	                #CambioReqVel := "Motore".M[#K_MotoreInt].Dati.VeloRichPerc <> "Motore".M[#K_MotoreInt].In.CmdVelocitaRich;
	                IF #CambioReqVel THEN
	                    "Motore".M[#K_MotoreInt].Dati.VeloRichPerc := "Motore".M[#K_MotoreInt].In.CmdVelocitaRich;
	                END_IF;
	(* Controllo Cambio Accelerazione richiesta *)
	                #CambioReqAcc := "Motore".M[#K_MotoreInt].Dati.AccRichPerc <> "Motore".M[#K_MotoreInt].In.Acc;
	                IF #CambioReqAcc THEN
	                    "Motore".M[#K_MotoreInt].Dati.AccRichPerc := "Motore".M[#K_MotoreInt].In.Acc;
	                END_IF;
	(* Controllo Cambio Decelerazione richiesta *)
	                #CambioReqDec := "Motore".M[#K_MotoreInt].Dati.DecRichPerc <> "Motore".M[#K_MotoreInt].In.Dec;
	                IF #CambioReqDec THEN
	                    "Motore".M[#K_MotoreInt].Dati.DecRichPerc := "Motore".M[#K_MotoreInt].In.Dec;
	                END_IF;
	            END_REGION
	            REGION Direzione Movimento Richiesta
	                IF "Motore".M[#K_MotoreInt].In.CmdPosRich AND "Motore".M[#K_MotoreInt].Out.Pronto AND #AbilDirPos THEN
	                    #ReqDirPos := TRUE;
	                    #ReqDirNeg := FALSE;
	                    #UnaDirezioneRichiesta := TRUE;
	                ELSIF "Motore".M[#K_MotoreInt].In.CmdNegRich AND "Motore".M[#K_MotoreInt].Out.Pronto AND #AbilDirNeg THEN
	                    #ReqDirPos := FALSE;
	                    #ReqDirNeg := TRUE;
	                    #UnaDirezioneRichiesta := TRUE;
	                ELSE
	                    #ReqDirPos := FALSE;
	                    #ReqDirNeg := FALSE;
	                    #UnaDirezioneRichiesta := FALSE;
	                END_IF;
	            END_REGION
	        END_IF;
	    END_REGION ;
	    REGION Parameter profile
	        REGION VelocitÃ  Minima
	            IF NOT "Motore".M[#K_MotoreInt].Dati.ActVelPos AND NOT "Motore".M[#K_MotoreInt].Dati.ActVelNeg AND #ReqDirNeg OR "Motore".M[#K_MotoreInt].Dati.ActVelNeg THEN
	                #SpazioFrenoDir := "Motore".M[#K_MotoreInt].Prm.SpazioArrestoNeg;
	                #VeloFrenoDir := "Motore".M[#K_MotoreInt].Prm.VelSgancioFrenoNeg;
	            ELSE
	                #SpazioFrenoDir := "Motore".M[#K_MotoreInt].Prm.SpazioArrestoPos;
	                #VeloFrenoDir := "Motore".M[#K_MotoreInt].Prm.VelSgancioFrenoPos;
	            END_IF;
	        END_REGION
	        REGION Controllo VelocitÃ
	(* Controllo che la velocitÃ  sia all'interno del limite Sgancio Freno < VeloRich < VeloMax *)
	            "Motore".M[#K_MotoreInt].Allarmi.TrgVelMinFreno := false;
	            "Motore".M[#K_MotoreInt].Allarmi.TrgVelMaxMax := false;
	            "Motore".M[#K_MotoreInt].Allarmi.TrgVelCamMinFreno := false;
	            "Motore".M[#K_MotoreInt].Allarmi.TrgVelCamMaxMax := false;
	            IF #UnaDirezioneRichiesta THEN
	                IF "Motore".M[#K_MotoreInt].Dati.VeloRichPerc < #VeloFrenoDir THEN
	                    "Motore".M[#K_MotoreInt].Allarmi.TrgVelMinFreno := true;
	                    "Motore".M[#K_MotoreInt].Allarmi.Parametri := TRUE;
	                    "Motore".M[#K_MotoreInt].Dati.VeloRichPerc := #VeloFrenoDir;
	                END_IF;
	                IF "Motore".M[#K_MotoreInt].Dati.VeloRichPerc > "Motore".M[#K_MotoreInt].Prm.C.VelMax THEN
	                    "Motore".M[#K_MotoreInt].Allarmi.TrgVelMaxMax := true;
	                    "Motore".M[#K_MotoreInt].Allarmi.Parametri := TRUE;
	                    "Motore".M[#K_MotoreInt].Dati.VeloRichPerc := "Motore".M[#K_MotoreInt].Prm.C.VelMax;
	                END_IF;
	                (* Controllo che la velocitÃ  di cambio VelocitÃ  sia all'interno del limite Sgancio Freno < VeloRich < VeloMax *)
	                IF "Motore".M[#K_MotoreInt].In.CambioVelDaPunto THEN
	                    "Motore".M[#K_MotoreInt].Dati.VeloDopoCambioRich := "Motore".M[#K_MotoreInt].In.VelCambioVel;
	                    IF "Motore".M[#K_MotoreInt].Dati.VeloDopoCambioRich < #VeloFrenoDir THEN
	                        "Motore".M[#K_MotoreInt].Allarmi.TrgVelCamMinFreno := true;
	                        "Motore".M[#K_MotoreInt].Allarmi.Parametri := TRUE;
	                        "Motore".M[#K_MotoreInt].Dati.VeloDopoCambioRich := #VeloFrenoDir;
	                    END_IF;
	                    IF "Motore".M[#K_MotoreInt].Dati.VeloDopoCambioRich > "Motore".M[#K_MotoreInt].Prm.C.VelMax THEN
	                        "Motore".M[#K_MotoreInt].Allarmi.TrgVelCamMaxMax := true;
	                        "Motore".M[#K_MotoreInt].Allarmi.Parametri := TRUE;
	                        "Motore".M[#K_MotoreInt].Dati.VeloDopoCambioRich := "Motore".M[#K_MotoreInt].Prm.C.VelMax;
	                    END_IF;
	                END_IF;
	            END_IF;
	        END_REGION
	        REGION Controllo Decelerazione di emergenza
	            IF "Motore".M[#K_MotoreInt].Dati.Memo_Req_Dec_Emergenza <> "Motore".M[#K_MotoreInt].Prm.DecEmergenza THEN
	                "Motore".M[#K_MotoreInt].Allarmi.DecEmergenzaRichZero := "Motore".M[#K_MotoreInt].Prm.DecEmergenza < 100;
	                IF "Motore".M[#K_MotoreInt].Allarmi.DecEmergenzaRichZero THEN
	                    "Motore".M[#K_MotoreInt].Dati.Memo_Req_Dec_Emergenza := 100;
	                    "Motore".M[#K_MotoreInt].Allarmi.Parametri := TRUE;
	                    #CambioReqAcc := true;
	                    #CambioReqDec := true;
	                ELSE
	                    "Motore".M[#K_MotoreInt].Dati.Memo_Req_Dec_Emergenza := "Motore".M[#K_MotoreInt].Prm.DecEmergenza;
	                END_IF;
	            END_IF;
	        END_REGION
	        REGION Controllo Decelerazione
	            IF #CambioReqDec THEN
	                "Motore".M[#K_MotoreInt].Allarmi.DecRichZero := "Motore".M[#K_MotoreInt].Dati.DecRichPerc < 100;
	                IF "Motore".M[#K_MotoreInt].Allarmi.DecRichZero THEN
	                    "Motore".M[#K_MotoreInt].Dati.DecRichPerc := 100;
	                    "Motore".M[#K_MotoreInt].Allarmi.Parametri := TRUE;
	                END_IF;
	                "Motore".M[#K_MotoreInt].Allarmi.DecRichMaxMaxDec := "Motore".M[#K_MotoreInt].Dati.DecRichPerc > "Motore".M[#K_MotoreInt].Dati.Memo_Req_Dec_Emergenza;
	                IF "Motore".M[#K_MotoreInt].Allarmi.DecRichMaxMaxDec THEN
	                    "Motore".M[#K_MotoreInt].Dati.DecRichPerc := "Motore".M[#K_MotoreInt].Dati.Memo_Req_Dec_Emergenza;
	                    "Motore".M[#K_MotoreInt].Allarmi.Parametri := TRUE;
	                END_IF;
	            END_IF;
	        END_REGION
	        REGION Controllo Decelerazione Finale
	            "Motore".M[#K_MotoreInt].Allarmi.DecFinaleRichZero := "Motore".M[#K_MotoreInt].Prm.DecFinale < 100;
	            IF "Motore".M[#K_MotoreInt].Allarmi.DecFinaleRichZero THEN
	                "Motore".M[#K_MotoreInt].Prm.DecFinale := 100;
	                "Motore".M[#K_MotoreInt].Allarmi.Parametri := TRUE;
	            END_IF;
	            "Motore".M[#K_MotoreInt].Allarmi.DecFinaleRichMaxMaxDec := "Motore".M[#K_MotoreInt].Prm.DecFinale > "Motore".M[#K_MotoreInt].Dati.Memo_Req_Dec_Emergenza;
	            IF "Motore".M[#K_MotoreInt].Allarmi.DecFinaleRichMaxMaxDec THEN
	                "Motore".M[#K_MotoreInt].Prm.DecFinale := "Motore".M[#K_MotoreInt].Dati.Memo_Req_Dec_Emergenza;
	                "Motore".M[#K_MotoreInt].Allarmi.Parametri := TRUE;
	            END_IF;
	            IF "Motore".M[#K_MotoreInt].Prm.DecFinale <> "Motore".M[#K_MotoreInt].Dati.DecReqFinaleInLavo THEN
	                IF NOT "Motore".M[#K_MotoreInt].Out.InMarcia OR "Motore".M[#K_MotoreInt].Prm.DecFinale > "Motore".M[#K_MotoreInt].Dati.DecReqFinaleInLavo THEN
	                    "Motore".M[#K_MotoreInt].Dati.DecReqFinaleInLavo := "Motore".M[#K_MotoreInt].Prm.DecFinale;
	                END_IF;
	            END_IF;
	        END_REGION
	        REGION Controllo Accelerazione
	            IF #CambioReqAcc THEN
	                "Motore".M[#K_MotoreInt].Allarmi.AccRichZero := "Motore".M[#K_MotoreInt].Dati.AccRichPerc < 100;
	                IF "Motore".M[#K_MotoreInt].Allarmi.AccRichZero THEN
	                    "Motore".M[#K_MotoreInt].Dati.AccRichPerc := 100;
	                    "Motore".M[#K_MotoreInt].Allarmi.Parametri := TRUE;
	                END_IF;
	                "Motore".M[#K_MotoreInt].Allarmi.AccRichMaxMaxDec := "Motore".M[#K_MotoreInt].Dati.AccRichPerc > "Motore".M[#K_MotoreInt].Dati.Memo_Req_Dec_Emergenza;
	                IF "Motore".M[#K_MotoreInt].Allarmi.AccRichMaxMaxDec THEN
	                    "Motore".M[#K_MotoreInt].Dati.AccRichPerc := "Motore".M[#K_MotoreInt].Dati.Memo_Req_Dec_Emergenza;
	                    "Motore".M[#K_MotoreInt].Allarmi.Parametri := TRUE;
	                END_IF;
	            END_IF;
	        END_REGION
	        REGION Assegnazione decelerazione
	            IF "Motore".M[#K_MotoreInt].Dati.DecRichPerc <> "Motore".M[#K_MotoreInt].Dati.DecReqInLavo THEN
	                IF NOT "Motore".M[#K_MotoreInt].Out.InMarcia OR "Motore".M[#K_MotoreInt].Dati.DecRichPerc > "Motore".M[#K_MotoreInt].Dati.DecReqInLavo OR "Motore".M[#K_MotoreInt].Out.VelAss < #VeloBassaConv THEN
	                    "Motore".M[#K_MotoreInt].Dati.DecReqInLavo := "Motore".M[#K_MotoreInt].Dati.DecRichPerc;
	                END_IF;
	            END_IF;
	        END_REGION
	        REGION Assegnazione decelerazione D'emergenza
	            IF "Motore".M[#K_MotoreInt].Dati.Memo_Req_Dec_Emergenza <> "Motore".M[#K_MotoreInt].Dati.DecReqEmergInLavo THEN
	                IF NOT "Motore".M[#K_MotoreInt].Out.InMarcia OR "Motore".M[#K_MotoreInt].Dati.Memo_Req_Dec_Emergenza > "Motore".M[#K_MotoreInt].Dati.DecReqEmergInLavo THEN
	                    "Motore".M[#K_MotoreInt].Dati.DecReqEmergInLavo := "Motore".M[#K_MotoreInt].Dati.Memo_Req_Dec_Emergenza;
	                END_IF;
	            END_IF;
	        END_REGION
	        REGION Calcolo Lo Spazio Di Arresto
	            #ReqDecBassa := FALSE;
	            #ReqDecStop := FALSE;
	            #BloccaAcc := FALSE;
	            IF "Motore".M[#K_MotoreInt].Out.InMarcia THEN
	                IF "Motore".M[#K_MotoreInt].Out.VelAss > #VeloBassaConv THEN
	                    #SpazioStop_01 := (SQR(IN := "Motore".M[#K_MotoreInt].Out.VelAss) - SQR(IN := #VeloBassaConv)) / DINT_TO_REAL("Motore".M[#K_MotoreInt].Dati.DecReqInLavo) / 2.0;
	                    #SpazioStop_02 := DINT_TO_REAL(IN := "Motore".M[#K_MotoreInt].Prm.TBassaVel) * #VeloBassaConv / 1000.0;
	                    #SpazioStop_03 := (SQR(IN := #VeloBassaConv) - SQR(IN := DINT_TO_REAL(#VeloFrenoDir))) / DINT_TO_REAL("Motore".M[#K_MotoreInt].Dati.DecReqFinaleInLavo) / 2.0;
	                ELSE
	                    #SpazioStop_01 := 0.0;
	                    #SpazioStop_02 := 0.0;
	                    #SpazioStop_03 := (SQR(IN := "Motore".M[#K_MotoreInt].Out.VelAss) - SQR(IN := DINT_TO_REAL(#VeloFrenoDir))) / DINT_TO_REAL("Motore".M[#K_MotoreInt].Dati.DecReqFinaleInLavo) / 2.0;
	                    ;
	                END_IF;
	                #SpazioStop_04 := INT_TO_REAL("Motore".M[#K_MotoreInt].Prm.TReazioneSistema) * ("Motore".M[#K_MotoreInt].Out.VelAss - DINT_TO_REAL(#VeloFrenoDir)) / 1000.0;
	                #SpazioStop := TRUNC(IN := #SpazioStop_03 + #SpazioStop_04) + #SpazioFrenoDir;
	                #SpazioBassa := TRUNC(IN := #SpazioStop_01 + #SpazioStop_02) + #SpazioStop;
	                IF #FunzPositioning THEN
	                    #BloccaAcc := TRUNC(("Motore".M[#K_MotoreInt].Out.VelAss * INT_TO_REAL("Motore".M[#K_MotoreInt].Prm.TMinVCost) / 1000.0)) + #SpazioStop > #DistTRG_ASS;
	                    #ReqDecBassa := #DistTRG_ASS < #SpazioBassa;
	                    #ReqDecStop := #DistTRG_ASS < #SpazioStop;
	                END_IF;
	            ELSE
	                #SpazioBassa := #SpazioStop := #SpazioFrenoDir;
	            END_IF;
	        END_REGION
	        REGION Calcolo lo spazio passaggio seconda Vel.
	            IF #FunzPositioning AND "Motore".M[#K_MotoreInt].In.CambioVelDaPunto AND NOT "Motore".M[#K_MotoreInt].Dati.MotoreFermo THEN
	                // Lo spazio di cambio velocitÃ  Ã¨ dato dalla somma dei seguenti fattori:

	                // 1) Spazio necessario al cambio velocitÃ  dell'asse calcolando una rampa trapezoidale.
	                // 2) Simulazione dello spazio percorso dall'asse durante la reazione del segnale analogico.

	                // Condizione 01 -Trapezio passaggio dalla velocitÃ  di lavoro alla velocitÃ  bassa
	                #SpazioCambioVel_01 := ("Motore".M[#K_MotoreInt].Out.VelAss ** 2 - DINT_TO_REAL("Motore".M[#K_MotoreInt].Dati.VeloDopoCambioRich) ** 2) / DINT_TO_REAL("Motore".M[#K_MotoreInt].Dati.DecReqInLavo) / 2.0;
	                #SpazioCambioVel_02 := INT_TO_REAL("Motore".M[#K_MotoreInt].Prm.TReazioneSistema) * "Motore".M[#K_MotoreInt].Out.VelAss / 1000.0;
	                #SpazioCambioVel := TRUNC(#SpazioCambioVel_01 + #SpazioCambioVel_02);
	                // Continua solo se cambio velocitÃ  Ã¨ attivo
	                // Calcolo la distanza dal cambio velocitÃ
	                IF NOT "Motore".M[#K_MotoreInt].In.PosRelativo THEN
	                    IF "Motore".M[#K_MotoreInt].Prm.Mech.EndLess THEN
	                        WHILE "Motore".M[#K_MotoreInt].In.PosCambioVel > "Motore".M[#K_MotoreInt].Prm.Enc.ModuloPosEnc DO
	                            "Motore".M[#K_MotoreInt].In.PosCambioVel -= #RicircoloTotale;
	                        END_WHILE;
	                        WHILE "Motore".M[#K_MotoreInt].In.PosCambioVel < "Motore".M[#K_MotoreInt].Prm.Enc.ModuloNegEnc DO
	                            "Motore".M[#K_MotoreInt].In.PosCambioVel += #RicircoloTotale;
	                        END_WHILE;
	                    END_IF;
	                    IF "Motore".M[#K_MotoreInt].Dati.ActVelPos THEN
	                        #DistCambioVel := "Motore".M[#K_MotoreInt].Out.ActPos + #SpazioCambioVel - "Motore".M[#K_MotoreInt].In.PosCambioVel;
	                    ELSE
	                        #DistCambioVel := "Motore".M[#K_MotoreInt].Out.ActPos - #SpazioCambioVel - "Motore".M[#K_MotoreInt].In.PosCambioVel;
	                    END_IF;
	                    IF "Motore".M[#K_MotoreInt].Prm.Mech.EndLess THEN
	                        IF #DistCambioVel > #MezzoRicircoloTotale THEN
	                            #DistCambioVel -= #RicircoloTotale;
	                        END_IF;
	                        IF #DistCambioVel < - #MezzoRicircoloTotale THEN
	                            #DistCambioVel += #RicircoloTotale;
	                        END_IF;
	                    END_IF;
	                    #ReqCambioVel := #DistCambioVel >= 0 AND "Motore".M[#K_MotoreInt].Dati.ActVelPos OR #DistCambioVel < 0 AND "Motore".M[#K_MotoreInt].Dati.ActVelNeg;
	                ELSE
	                    #ReqCambioVel := "Motore".M[#K_MotoreInt].Dati.MovRelRichiesto - #DistTRG_ASS + #SpazioCambioVel > "Motore".M[#K_MotoreInt].In.PosCambioVel;
	                END_IF;
	            ELSE
	                #ReqCambioVel := FALSE;
	                #SpazioCambioVel := 0;
	            END_IF;

	        END_REGION
	        REGION Pos.Motore + Spazio Arresto
	            IF "Motore".M[#K_MotoreInt].Out.InMarcia THEN
	                "Motore".M[#K_MotoreInt].Out.SpazioStop := #SpazioBassa;
	                IF "Motore".M[#K_MotoreInt].Dati.ActVelPos THEN
	                    "Motore".M[#K_MotoreInt].Out.ActPosPiuStop := "Motore".M[#K_MotoreInt].Out.ActPos + #SpazioBassa;
	                ELSE
	                    "Motore".M[#K_MotoreInt].Out.ActPosPiuStop := "Motore".M[#K_MotoreInt].Out.ActPos - #SpazioBassa;
	                END_IF;
	                IF "Motore".M[#K_MotoreInt].Prm.Mech.EndLess THEN
	                    IF "Motore".M[#K_MotoreInt].Out.ActPosPiuStop < "Motore".M[#K_MotoreInt].Prm.Enc.ModuloNegEnc THEN
	                        "Motore".M[#K_MotoreInt].Out.ActPosPiuStop += #RicircoloTotale;
	                    END_IF;
	                    IF "Motore".M[#K_MotoreInt].Out.ActPosPiuStop > "Motore".M[#K_MotoreInt].Prm.Enc.ModuloPosEnc THEN
	                        "Motore".M[#K_MotoreInt].Out.ActPosPiuStop -= #RicircoloTotale;
	                    END_IF;
	                END_IF;
	            ELSE
	                "Motore".M[#K_MotoreInt].Out.ActPosPiuStop := "Motore".M[#K_MotoreInt].Out.ActPos;
	                "Motore".M[#K_MotoreInt].Out.SpazioStop := 0;
	            END_IF;
	        END_REGION
	    END_REGION ;
	    REGION Delay brake
	        REGION Ritrado Aggancio/Sgancio Freno
	            IF "Motore".M[#K_MotoreInt].Prm.FrenoPresente THEN
	                IF "Motore".M[#K_MotoreInt].Prm.FBKFrenoPresente THEN
	                    "Motore".M[#K_MotoreInt].Dati.StatoFreno := "Motore".M[#K_MotoreInt].In.FrenoSganciato;
	                ELSE
	                    "Motore".M[#K_MotoreInt].Dati.StatoFreno := "Motore".M[#K_MotoreInt].Out.CmdFreno;
	                END_IF;
	                IF "Motore".M[#K_MotoreInt].Dati.StatoFreno THEN
	                    "Motore".M[#K_MotoreInt].Dati.ContAggancioFreno := 0;
	                    "Motore".M[#K_MotoreInt].Dati.RitAggancioFreno := false;
	                    IF NOT "Motore".M[#K_MotoreInt].Out.RitSgancioFreno THEN
	                        "Motore".M[#K_MotoreInt].Out.RitSgancioFreno := "Motore".M[#K_MotoreInt].Dati.ContSgancioFreno >= "Motore".M[#K_MotoreInt].Prm.TSgancioFreno;
	                        "Motore".M[#K_MotoreInt].Dati.ContSgancioFreno += REAL_TO_INT("Zona".Comuni.TempoCicloCpu_r);
	                    END_IF;
	                ELSE
	                    "Motore".M[#K_MotoreInt].Dati.ContSgancioFreno := 0;
	                    "Motore".M[#K_MotoreInt].Out.RitSgancioFreno := false;
	                    IF NOT "Motore".M[#K_MotoreInt].Dati.RitAggancioFreno THEN
	                        "Motore".M[#K_MotoreInt].Dati.RitAggancioFreno := "Motore".M[#K_MotoreInt].Dati.ContAggancioFreno >= "Motore".M[#K_MotoreInt].Prm.TAggancioFreno;
	                        "Motore".M[#K_MotoreInt].Dati.ContAggancioFreno += REAL_TO_INT("Zona".Comuni.TempoCicloCpu_r);
	                    END_IF;
	                END_IF;
	            ELSE
	                "Motore".M[#K_MotoreInt].Out.RitSgancioFreno := "Motore".M[#K_MotoreInt].Out.CmdFreno;
	                "Motore".M[#K_MotoreInt].Dati.RitAggancioFreno := NOT "Motore".M[#K_MotoreInt].Out.RitSgancioFreno;
	            END_IF;
	        END_REGION
	        REGION Premagnetizzazione
	            IF "Motore".M[#K_MotoreInt].Dati.MotoreFermo THEN
	                "Motore".M[#K_MotoreInt].Prm.C.ContPrema := 0;
	                "Motore".M[#K_MotoreInt].Out.PremaOK := false;
	            ELSIF NOT "Motore".M[#K_MotoreInt].Out.PremaOK THEN
	                IF "Motore".M[#K_MotoreInt].Prm.VelPrema <= 0 OR "Motore".M[#K_MotoreInt].Prm.VelPrema > #VeloFrenoDir THEN
	                    "Motore".M[#K_MotoreInt].Prm.VelPrema := #VeloFrenoDir;
	                END_IF;
	                "Motore".M[#K_MotoreInt].Prm.C.ContPrema += REAL_TO_INT("Zona".Comuni.TempoCicloCpu_r);
	                "Motore".M[#K_MotoreInt].Out.PremaOK := "Motore".M[#K_MotoreInt].Prm.C.ContPrema > "Motore".M[#K_MotoreInt].Prm.TPrema;
	            END_IF;
	        END_REGION

	        IF "Motore".M[#K_MotoreInt].Out.PremaOK AND "Motore".M[#K_MotoreInt].Out.RitSgancioFreno AND #UnaDirezioneRichiesta THEN
	            "Motore".M[#K_MotoreInt].Out.InMarcia := true;
	        ELSIF "Motore".M[#K_MotoreInt].Dati.RitAggancioFreno THEN
	            "Motore".M[#K_MotoreInt].Out.InMarcia := false;
	        END_IF;
	        REGION TimeOut Premagnetizzazione
	            IF "Motore".M[#K_MotoreInt].In.Premagnetizza AND NOT "Motore".M[#K_MotoreInt].Out.InMarcia THEN
	                IF NOT "Zona".Z[#K_ZonaInt].Out.Auto OR NOT "Zona".Z[#K_Zona].Out.CentralinaOk OR "Motore".M[#K_MotoreInt].Out.Allarme OR "Motore".M[#K_MotoreInt].In.DriverFault THEN
	                    "Motore".M[#K_MotoreInt].In.Premagnetizza := "Motore".M[#K_MotoreInt].In.PremagnetizzaPos := "Motore".M[#K_MotoreInt].In.PremagnetizzaNeg := false;
	                END_IF;
	                IF "Motore".M[#K_MotoreInt].Prm.VelPrema <> 1 THEN
	                    "Motore".M[#K_MotoreInt].Prm.PremaNoFreno := false;
	                END_IF;
	                "Motore".M[#K_MotoreInt].Prm.TOutPrema := MAX(IN1 := "Motore".M[#K_MotoreInt].Prm.TOutPrema, IN2 := "Motore".M[#K_MotoreInt].Prm.TPrema + 50);
	                IF NOT "Motore".M[#K_MotoreInt].Out.InMarcia THEN
	                    "Motore".M[#K_MotoreInt].Out.TOUTPrema := "Motore".M[#K_MotoreInt].Dati.ContTimeOutPrema > "Motore".M[#K_MotoreInt].Prm.TOutPrema;
	                    IF NOT "Motore".M[#K_MotoreInt].Out.TOUTPrema THEN
	                        "Motore".M[#K_MotoreInt].Dati.ContTimeOutPrema += REAL_TO_INT("Zona".Comuni.TempoCicloCpu_r);
	                    END_IF;
	                ELSE
	                    "Motore".M[#K_MotoreInt].Dati.ContTimeOutPrema := 0;
	                END_IF;
	            ELSE
	                "Motore".M[#K_MotoreInt].Dati.ContTimeOutPrema := 0;
	                "Motore".M[#K_MotoreInt].Out.TOUTPrema := false;
	            END_IF;
	        END_REGION
	    END_REGION ;
	    REGION Request speed and brake command
	        #ReqStop := NOT #UnaDirezioneRichiesta;
	        IF (#ReqDirPos AND "Motore".M[#K_MotoreInt].Dati.ActVelNeg) OR (#ReqDirNeg AND "Motore".M[#K_MotoreInt].Dati.ActVelPos) THEN
	            #ReqStop := true;
	            "Motore".M[#K_MotoreInt].Dati.ContAbilAccDopoCambioDir := "Motore".M[#K_MotoreInt].Prm.TReazioneSistema;
	        ELSIF "Motore".M[#K_MotoreInt].Dati.ContAbilAccDopoCambioDir > 0 THEN
	            "Motore".M[#K_MotoreInt].Dati.ContAbilAccDopoCambioDir -= REAL_TO_INT("Zona".Comuni.TempoCicloCpu_r);
	        END_IF;
	        IF NOT #ReqStop AND NOT #ReqDecStop THEN
	            IF NOT "Motore".M[#K_MotoreInt].Out.PremaOK AND NOT "Motore".M[#K_MotoreInt].Out.InMarcia THEN
	                "Motore".M[#K_MotoreInt].Dati.VeloMinConv := DINT_TO_REAL("Motore".M[#K_MotoreInt].Prm.VelPrema);
	            ELSE
	                "Motore".M[#K_MotoreInt].Dati.VeloMinConv := DINT_TO_REAL(#VeloFrenoDir);
	            END_IF;
	            IF NOT "Motore".M[#K_MotoreInt].Out.InMarcia THEN
	                "Motore".M[#K_MotoreInt].Dati.ReqVelConv := "Motore".M[#K_MotoreInt].Dati.VeloMinConv;
	            ELSIF #ReqDecBassa THEN
	                "Motore".M[#K_MotoreInt].Dati.ReqVelConv := #VeloBassaConv;
	            ELSIF NOT #ReqCambioVel THEN
	                "Motore".M[#K_MotoreInt].Dati.ReqVelConv := DINT_TO_REAL("Motore".M[#K_MotoreInt].Dati.VeloRichPerc);
	            ELSE
	                "Motore".M[#K_MotoreInt].Dati.ReqVelConv := DINT_TO_REAL(MIN(IN1 := "Motore".M[#K_MotoreInt].Dati.VeloDopoCambioRich, IN2 := "Motore".M[#K_MotoreInt].Dati.VeloRichPerc));
	            END_IF;
	            "Motore".M[#K_MotoreInt].Out.FaseDec := "Motore".M[#K_MotoreInt].Dati.ReqVelConv < "Motore".M[#K_MotoreInt].Out.VelAss;
	        ELSE
	            "Motore".M[#K_MotoreInt].Out.FaseDec := TRUE;
	        END_IF;
	        IF NOT "Motore".M[#K_MotoreInt].Out.FaseDec THEN
	            "Motore".M[#K_MotoreInt].Out.FaseAcc := NOT #BloccaAcc AND "Motore".M[#K_MotoreInt].Dati.ReqVelConv > "Motore".M[#K_MotoreInt].Out.VelAss AND "Motore".M[#K_MotoreInt].Dati.ContAbilAccDopoCambioDir <= 0;
	            IF "Motore".M[#K_MotoreInt].Out.FaseAcc THEN
	                // Calcolo Accelerazione
	                "Motore".M[#K_MotoreInt].Out.VelAss += DINT_TO_REAL("Motore".M[#K_MotoreInt].Dati.AccRichPerc) * INT_TO_REAL(REAL_TO_INT("Zona".Comuni.TempoCicloCpu_r)) / 1000.0;
	                "Motore".M[#K_MotoreInt].Out.VelAss := LIMIT(MN := "Motore".M[#K_MotoreInt].Dati.VeloMinConv, IN := "Motore".M[#K_MotoreInt].Out.VelAss, MX := "Motore".M[#K_MotoreInt].Dati.ReqVelConv);
	            END_IF;
	        ELSE
	            "Motore".M[#K_MotoreInt].Out.FaseAcc := false;
	            // Calcolo Decelerazione
	            IF NOT "Motore".M[#K_MotoreInt].Dati.MotoreFermo THEN
	                (* Seleziono la Decelerazione con cui devo lavorare *)
	                IF NOT "Motore".M[#K_MotoreInt].Out.Pronto THEN
	                    #DecActRich := "Motore".M[#K_MotoreInt].Dati.DecReqEmergInLavo;
	                ELSIF "Motore".M[#K_MotoreInt].Out.VelAss > #VeloBassaConv THEN
	                    #DecActRich := "Motore".M[#K_MotoreInt].Dati.DecReqInLavo;
	                ELSE
	                    #DecActRich := "Motore".M[#K_MotoreInt].Dati.DecReqFinaleInLavo;
	                END_IF;
	                "Motore".M[#K_MotoreInt].Out.VelAss -= DINT_TO_REAL(#DecActRich) * INT_TO_REAL(REAL_TO_INT("Zona".Comuni.TempoCicloCpu_r)) / 1000.0;
	                "Motore".M[#K_MotoreInt].Out.VelAss := MAX(IN1 := "Motore".M[#K_MotoreInt].Dati.VeloMinConv, IN2 := "Motore".M[#K_MotoreInt].Out.VelAss);
	                // Forzo l'arresto se sono in zona di arresto
	                IF #ReqStop AND "Motore".M[#K_MotoreInt].Out.VelAss <= "Motore".M[#K_MotoreInt].Dati.VeloMinConv THEN
	                    IF "Motore".M[#K_MotoreInt].Prm.CambioDirNoFreno THEN
	                        IF "Motore".M[#K_MotoreInt].Dati.ActVelPos AND #ReqDirNeg THEN
	                            "Motore".M[#K_MotoreInt].Dati.ActVelPos := false;
	                            "Motore".M[#K_MotoreInt].Dati.ActVelNeg := true;
	                            #ReqStop := false;
	                            "Motore".M[#K_MotoreInt].Dati.CambioDirezioneAlVolo := true;
	                        ELSIF "Motore".M[#K_MotoreInt].Dati.ActVelNeg AND #ReqDirPos THEN
	                            "Motore".M[#K_MotoreInt].Dati.ActVelPos := true;
	                            "Motore".M[#K_MotoreInt].Dati.ActVelNeg := false;
	                            #ReqStop := false;
	                            "Motore".M[#K_MotoreInt].Dati.CambioDirezioneAlVolo := true;
	                        ELSE
	                            "Motore".M[#K_MotoreInt].Dati.CambioDirezioneAlVolo := false;
	                        END_IF;
	                    END_IF;
	                    IF NOT "Motore".M[#K_MotoreInt].Dati.CambioDirezioneAlVolo THEN
	                        IF "Motore".M[#K_MotoreInt].Dati.RitAggancioFreno OR "Motore".M[#K_MotoreInt].Allarmi.Freno OR "Motore".M[#K_MotoreInt].Allarmi.Freno2 THEN
	                            "Motore".M[#K_MotoreInt].Out.VelAss := 0.0;
	                        ELSE
	                            "Motore".M[#K_MotoreInt].Out.VelAss := DINT_TO_REAL("Motore".M[#K_MotoreInt].Prm.VelPrema);
	                        END_IF;
	                    END_IF;
	                END_IF;
	            END_IF;
	        END_IF;
	        REGION Gestione Direzione Del Movimento
	            IF "Motore".M[#K_MotoreInt].Dati.MotoreFermo AND #ReqDirPos OR "Motore".M[#K_MotoreInt].Dati.ActVelPos THEN
	                "Motore".M[#K_MotoreInt].Out.Vel := "Motore".M[#K_MotoreInt].Out.VelAss;
	            ELSIF "Motore".M[#K_MotoreInt].Dati.MotoreFermo AND #ReqDirNeg OR "Motore".M[#K_MotoreInt].Dati.ActVelNeg THEN
	                "Motore".M[#K_MotoreInt].Out.Vel := - "Motore".M[#K_MotoreInt].Out.VelAss;
	            END_IF;
	        END_REGION
	        REGION Velo Premagnetizzazione
	            IF NOT "Motore".M[#K_MotoreInt].Out.InMarcia THEN
	                IF "Motore".M[#K_MotoreInt].In.Premagnetizza THEN
	                    IF NOT "Motore".M[#K_MotoreInt].Out.TOUTPrema AND NOT #UnaDirezioneRichiesta THEN
	                        IF "Motore".M[#K_MotoreInt].In.PremagnetizzaPos THEN
	                            "Motore".M[#K_MotoreInt].Out.VelAss := DINT_TO_REAL("Motore".M[#K_MotoreInt].Prm.VelPrema);
	                            "Motore".M[#K_MotoreInt].Out.Vel := "Motore".M[#K_MotoreInt].Out.VelAss;
	                        ELSIF "Motore".M[#K_MotoreInt].In.PremagnetizzaNeg THEN
	                            "Motore".M[#K_MotoreInt].Out.VelAss := DINT_TO_REAL("Motore".M[#K_MotoreInt].Prm.VelPrema);
	                            "Motore".M[#K_MotoreInt].Out.Vel := - "Motore".M[#K_MotoreInt].Out.VelAss;
	                        ELSIF "Motore".M[#K_MotoreInt].Out.RichMovPos THEN
	                            "Motore".M[#K_MotoreInt].Out.VelAss := DINT_TO_REAL("Motore".M[#K_MotoreInt].Prm.VelPrema);
	                            "Motore".M[#K_MotoreInt].Out.Vel := "Motore".M[#K_MotoreInt].Out.VelAss;
	                        ELSIF "Motore".M[#K_MotoreInt].Out.RichMovNeg THEN
	                            "Motore".M[#K_MotoreInt].Out.VelAss := DINT_TO_REAL("Motore".M[#K_MotoreInt].Prm.VelPrema);
	                            "Motore".M[#K_MotoreInt].Out.Vel := - "Motore".M[#K_MotoreInt].Out.VelAss;
	                        END_IF;
	                    END_IF;
	                END_IF;
	            END_IF;
	        END_REGION
	        REGION Controllo Direzione Motore
	            IF "Motore".M[#K_MotoreInt].Out.Vel > 0.0 THEN
	                "Motore".M[#K_MotoreInt].Dati.ActVelPos := TRUE;
	                "Motore".M[#K_MotoreInt].Dati.ActVelNeg := FALSE;
	                "Motore".M[#K_MotoreInt].Dati.MotoreFermo := FALSE;
	            ELSIF "Motore".M[#K_MotoreInt].Out.Vel < 0.0 THEN
	                "Motore".M[#K_MotoreInt].Dati.ActVelPos := FALSE;
	                "Motore".M[#K_MotoreInt].Dati.ActVelNeg := TRUE;
	                "Motore".M[#K_MotoreInt].Dati.MotoreFermo := FALSE;
	            ELSE
	                "Motore".M[#K_MotoreInt].Dati.ActVelPos := FALSE;
	                "Motore".M[#K_MotoreInt].Dati.ActVelNeg := FALSE;
	                "Motore".M[#K_MotoreInt].Dati.MotoreFermo := TRUE;
	            END_IF;
	            IF NOT "Motore".M[#K_MotoreInt].Prm.Mech.Direction THEN
	                "Motore".M[#K_MotoreInt].Out.CmdPosMotore := "Motore".M[#K_MotoreInt].Dati.ActVelPos;
	                "Motore".M[#K_MotoreInt].Out.CmdNegMotore := "Motore".M[#K_MotoreInt].Dati.ActVelNeg;
	            ELSE
	                "Motore".M[#K_MotoreInt].Out.CmdPosMotore := "Motore".M[#K_MotoreInt].Dati.ActVelNeg;
	                "Motore".M[#K_MotoreInt].Out.CmdNegMotore := "Motore".M[#K_MotoreInt].Dati.ActVelPos;
	            END_IF;
	            IF "Motore".M[#K_MotoreInt].Out.InMarcia THEN
	                "Motore".M[#K_MotoreInt].Out.ActDirPos := "Motore".M[#K_MotoreInt].Dati.ActVelPos;
	                "Motore".M[#K_MotoreInt].Out.ActDirNeg := "Motore".M[#K_MotoreInt].Dati.ActVelNeg;
	            ELSE
	                "Motore".M[#K_MotoreInt].Out.ActDirNeg := "Motore".M[#K_MotoreInt].Out.ActDirPos := false;
	            END_IF;
	        END_REGION
	        REGION GestioneFreno
	            IF #UnaDirezioneRichiesta AND "Motore".M[#K_MotoreInt].Out.PremaOK OR "Motore".M[#K_MotoreInt].Out.InMarcia THEN
	                #RichCmdFreno := (NOT #ReqStop AND "Motore".M[#K_MotoreInt].Out.VelAss = "Motore".M[#K_MotoreInt].Dati.VeloMinConv OR "Motore".M[#K_MotoreInt].Out.VelAss > "Motore".M[#K_MotoreInt].Dati.VeloMinConv);
	            ELSE
	                IF "Motore".M[#K_MotoreInt].Prm.PremaNoFreno THEN
	                    #RichCmdFreno := "Motore".M[#K_MotoreInt].Out.PremaOK AND NOT "Motore".M[#K_MotoreInt].Out.TOUTPrema AND "Motore".M[#K_MotoreInt].Out.VelAss = 1.0;
	                ELSE
	                    #RichCmdFreno := false;
	                END_IF;
	            END_IF;
	            IF #RichCmdFreno THEN
	                REGION Tempo Off Inverter Pronto
	                    IF "Motore".M[#K_MotoreInt].In.MotoreRun AND "Motore".M[#K_MotoreInt].Out.CmdFreno THEN
	                        "Motore".M[#K_MotoreInt].Dati.TOffInverterStatus := true;
	                        "Motore".M[#K_MotoreInt].Dati.ContTOffInverterStatus := 250;
	                    ELSIF "Motore".M[#K_MotoreInt].Dati.TOffInverterStatus THEN
	                        "Motore".M[#K_MotoreInt].Dati.ContTOffInverterStatus -= REAL_TO_INT("Zona".Comuni.TempoCicloCpu_r);
	                        "Motore".M[#K_MotoreInt].Dati.TOffInverterStatus := "Motore".M[#K_MotoreInt].Dati.ContTOffInverterStatus > 0;
	                    END_IF;
	                END_REGION
	                "Motore".M[#K_MotoreInt].Out.CmdFreno := ("Motore".M[#K_MotoreInt].Out.Pronto AND "Motore".M[#K_MotoreInt].Dati.TOffInverterStatus OR "Motore".M[#K_MotoreInt].In.MotoreRun) AND ("Motore".M[#K_MotoreInt].Dati.ActVelPos OR "Motore".M[#K_MotoreInt].Dati.ActVelNeg);
	            ELSE
	                "Motore".M[#K_MotoreInt].Out.CmdFreno := FALSE;
	            END_IF;
	        END_REGION
	    END_REGION ;
	    REGION Allarms, siren, lamp
	        REGION Controllo Allarmi Presenti
	            IF "Motore".M[#K_MotoreInt].Allarmi.Freno2 OR
	                "Motore".M[#K_MotoreInt].Allarmi.EncMismatch THEN
	                "Motore".M[#K_MotoreInt].Out.DisContattori := true;
	                "Motore".M[#K_MotoreInt].Out.Allarme := true;
	            ELSE
	                "Motore".M[#K_MotoreInt].Out.DisContattori := false;
	                IF "Motore".M[#K_MotoreInt].Allarmi.TOutMarcia OR
	                    "Motore".M[#K_MotoreInt].Allarmi.Freno OR
	                    "Motore".M[#K_MotoreInt].Allarmi.ConteggioEnc OR
	                    "Motore".M[#K_MotoreInt].Allarmi.Bloccato OR
	                    "Motore".M[#K_MotoreInt].Allarmi.TroppoVeloce OR
	                    "Motore".M[#K_MotoreInt].Allarmi.FolError OR
	                    "Motore".M[#K_MotoreInt].Allarmi.Direzione OR
	                    "Motore".M[#K_MotoreInt].Allarmi.TOUTMovimento OR
	                    "Motore".M[#K_MotoreInt].Allarmi.TOUT_Azzeramento OR
	                    "Motore".M[#K_MotoreInt].Allarmi.SezAperto OR
	                    "Motore".M[#K_MotoreInt].Allarmi.InverterFault OR
	                    "Motore".M[#K_MotoreInt].Allarmi.ComunInverter OR
	                    "Motore".M[#K_MotoreInt].Allarmi.ComunEncoder OR
	                    "Motore".M[#K_MotoreInt].Allarmi.TermicoVentola OR
	                    "Motore".M[#K_MotoreInt].Allarmi.RotturaCinghia OR
	                    "Motore".M[#K_MotoreInt].Allarmi.TimeOutAnticaduta OR
	                    "Motore".M[#K_MotoreInt].Allarmi.SpinaSicNoInPos
	                THEN
	                    "Motore".M[#K_MotoreInt].Out.Allarme := true;
	                ELSE
	                    "Motore".M[#K_MotoreInt].Out.Allarme := false;
	                END_IF;
	            END_IF;

	        END_REGION
	        REGION Gestione del reset, Lampada e Sirena
	            IF "Zona".Z[#K_ZonaInt].Gen.Reset THEN
	                IF NOT "Motore".M[#K_MotoreInt].Out.Sirena THEN
	                    IF "Motore".M[#K_MotoreInt].Allarmi.EncMismatch THEN
	                        "Motore".M[#K_MotoreInt].Dati.PosizioneAlloStop := "Motore".M[#K_MotoreInt].Out.ActPos;
	                    END_IF;
	                    IF "Motore".M[#K_MotoreInt].Allarmi.Direzione THEN
	                        "Motore".M[#K_MotoreInt].Dati.MemoCheckInversione := 0;
	                    END_IF;

	                    "Motore".M[#K_MotoreInt].Allarmi.TOutMarcia := false;
	                    "Motore".M[#K_MotoreInt].Allarmi.Freno := false;
	                    "Motore".M[#K_MotoreInt].Allarmi.Freno2 := false;
	                    "Motore".M[#K_MotoreInt].Allarmi.ConteggioEnc := false;
	                    "Motore".M[#K_MotoreInt].Allarmi.FolError := false;
	                    "Motore".M[#K_MotoreInt].Allarmi.Bloccato := false;
	                    "Motore".M[#K_MotoreInt].Allarmi.TroppoVeloce := false;
	                    "Motore".M[#K_MotoreInt].Allarmi.Direzione := false;
	                    "Motore".M[#K_MotoreInt].Allarmi.EncMismatch := false;
	                    "Motore".M[#K_MotoreInt].Allarmi.TOUTMovimento := false;
	                    "Motore".M[#K_MotoreInt].Allarmi.TOUT_Azzeramento := false;
	                    "Motore".M[#K_MotoreInt].Allarmi.InverterFault := false;
	                    "Motore".M[#K_MotoreInt].Allarmi.ComunInverter := false;
	                    "Motore".M[#K_MotoreInt].Allarmi.ComunEncoder := false;
	                    "Motore".M[#K_MotoreInt].Allarmi.TermicoVentola := false;
	                    "Motore".M[#K_MotoreInt].Allarmi.RotturaCinghia := false;
	                    "Motore".M[#K_MotoreInt].Allarmi.TimeOutAnticaduta := false;
	                    "Motore".M[#K_MotoreInt].Allarmi.SpinaSicNoInPos := false;
	                END_IF;
	                "Motore".M[#K_MotoreInt].Out.Sirena := false;
	            END_IF;
	        END_REGION
	        REGION TimeOut Marcia Motore
	            IF NOT "Motore".M[#K_MotoreInt].Dati.MotoreFermo AND NOT "Motore".M[#K_MotoreInt].In.MotoreRun AND NOT "Motore".M[#K_MotoreInt].Allarmi.TOutMarcia AND NOT "Motore".M[#K_MotoreInt].In.DriverFault THEN
	                "Motore".M[#K_MotoreInt].Dati.ContTimeOutInverter += REAL_TO_INT("Zona".Comuni.TempoCicloCpu_r);
	                IF "Motore".M[#K_MotoreInt].Dati.ContTimeOutInverter > 500 THEN
	                    "Motore".M[#K_MotoreInt].Allarmi.TOutMarcia := true;
	                END_IF;
	            ELSE
	                "Motore".M[#K_MotoreInt].Dati.ContTimeOutInverter := 0;
	            END_IF;

	        END_REGION
	        REGION Allarmi Freno
	            IF "Motore".M[#K_MotoreInt].Prm.FrenoPresente THEN
	                IF "Motore".M[#K_MotoreInt].Prm.FBKFrenoPresente THEN
	                    REGION Gestione del Time Out Freno 1 (Rilascio)
	                        IF "Motore".M[#K_MotoreInt].Out.CmdFreno AND NOT "Motore".M[#K_MotoreInt].Dati.StatoFreno AND NOT "Motore".M[#K_MotoreInt].Allarmi.Freno THEN
	                            "Motore".M[#K_MotoreInt].Dati.ContTimeOutFreno1 += REAL_TO_INT("Zona".Comuni.TempoCicloCpu_r);
	                            "Motore".M[#K_MotoreInt].Allarmi.Freno := "Motore".M[#K_MotoreInt].Dati.ContTimeOutFreno1 > 500;
	                        ELSE
	                            "Motore".M[#K_MotoreInt].Dati.ContTimeOutFreno1 := 0;
	                        END_IF;
	                    END_REGION
	                    REGION Gestione del Time Out Freno 2 (Aggancio)
	                        // Statement section REGION
	                        IF NOT "Motore".M[#K_MotoreInt].Out.CmdFreno THEN
	                            IF "Motore".M[#K_MotoreInt].Dati.ContTimeOutFreno2 < 150 THEN
	                                "Motore".M[#K_MotoreInt].Dati.ContTimeOutFreno2 += REAL_TO_INT("Zona".Comuni.TempoCicloCpu_r);
	                            ELSIF "Motore".M[#K_MotoreInt].Dati.StatoFreno THEN
	                                "Motore".M[#K_MotoreInt].Allarmi.Freno2 := TRUE;
	                            END_IF;
	                        ELSE
	                            "Motore".M[#K_MotoreInt].Dati.ContTimeOutFreno2 := 0;
	                        END_IF;
	                    END_REGION
	                END_IF;
	            END_IF;
	        END_REGION
	        REGION AllarmiEncoder
	            IF NOT "Motore".M[#K_MotoreInt].Prm.Enc.EncoderLess THEN
	                REGION Aggiornamento Stati Con Motore Fermo
	                    IF NOT "Motore".M[#K_MotoreInt].Out.InMarcia OR "Motore".M[#K_MotoreInt].Dati.CambioDirezioneAlVolo THEN
	                        "Motore".M[#K_MotoreInt].Dati.CambioDirezioneAlVolo := false;
	                        "Motore".M[#K_MotoreInt].Dati.TrgPosDint := "Motore".M[#K_MotoreInt].Dati.OldTrgPosDint := "Motore".M[#K_MotoreInt].Out.ActPos;
	                        "Motore".M[#K_MotoreInt].Prm.C.TrgPos := "Motore".M[#K_MotoreInt].Prm.C.EncPos;
	                        "Motore".M[#K_MotoreInt].Dati.ChFol_SpazioTarget := "Motore".M[#K_MotoreInt].Dati.ChFol_SpazioEncoder := 0;
	                        "Motore".M[#K_MotoreInt].Dati.ContCheckFollowError := 0;
	                    END_IF;
	                END_REGION
	                REGION Allarme conteggio Encoder
	                    // Se lo spazio percorso nell'ultimo ciclo programma dell'encoder Ã¨ 20 volte superiore
	                    // Allo spazio teorico per la velocitÃ  richiesta
	                    IF NOT #REQSetup THEN
	                        IF "Motore".M[#K_MotoreInt].Out.SpazioCicloEnc > "Motore".M[#K_MotoreInt].Prm.C.VelMax * REAL_TO_INT("Zona".Comuni.TempoCicloCpu_r) / 50 THEN
	                            "Motore".M[#K_MotoreInt].Allarmi.ConteggioEnc := true;
	                        END_IF;
	                    END_IF;
	                END_REGION
	                REGION Allarme d'inseguimento
	                    #AppoMoltPrecisione := "Motore".M[#K_MotoreInt].Prm.Precisione * 10;
	                    IF "Motore".M[#K_MotoreInt].Out.InMarcia AND NOT "Motore".M[#K_MotoreInt].Allarmi.FolError AND NOT "Motore".M[#K_MotoreInt].Allarmi.Bloccato AND NOT "Motore".M[#K_MotoreInt].Allarmi.TroppoVeloce THEN
	                        "Motore".M[#K_MotoreInt].Out.FollowingError := "Motore".M[#K_MotoreInt].Out.ActPos - "Motore".M[#K_MotoreInt].Dati.TrgPosDint;
	                        IF "Motore".M[#K_MotoreInt].Dati.ContCheckFollowError > 500 THEN
	                            "Motore".M[#K_MotoreInt].Dati.ChFol_SpazioTarget := ABS("Motore".M[#K_MotoreInt].Dati.ChFol_SpazioTarget);
	                            IF "Motore".M[#K_MotoreInt].Dati.ChFol_SpazioTarget > #AppoMoltPrecisione THEN
	                                "Motore".M[#K_MotoreInt].Dati.ChFol_SpazioEncoder := ABS("Motore".M[#K_MotoreInt].Dati.ChFol_SpazioEncoder);
	                                IF "Motore".M[#K_MotoreInt].Dati.ChFol_SpazioEncoder / 5 > "Motore".M[#K_MotoreInt].Dati.ChFol_SpazioTarget THEN
	                                    "Motore".M[#K_MotoreInt].Allarmi.TroppoVeloce := true;
	                                ELSIF "Motore".M[#K_MotoreInt].Dati.ChFol_SpazioEncoder * 5 < "Motore".M[#K_MotoreInt].Dati.ChFol_SpazioTarget THEN
	                                    IF NOT "Motore".M[#K_MotoreInt].Dati.MotorStop THEN
	                                        IF "Motore".M[#K_MotoreInt].Dati.AlmBloccato_Cont >= "NResetBloccato" THEN
	                                            "Motore".M[#K_MotoreInt].Allarmi.Bloccato := true;
	                                        ELSE
	                                            "Motore".M[#K_MotoreInt].Dati.AlmBloccato_Cont += 1;
	                                            "Motore".M[#K_MotoreInt].Dati.MotorStop := true;
	                                        END_IF;
	                                    END_IF;
	                                END_IF;
	                            END_IF;
	                            "Motore".M[#K_MotoreInt].Dati.ContCheckFollowError := 0;
	                            "Motore".M[#K_MotoreInt].Dati.ChFol_SpazioEncoder := "Motore".M[#K_MotoreInt].Dati.ChFol_SpazioTarget := 0;
	                        ELSE
	                            "Motore".M[#K_MotoreInt].Dati.ChFol_SpazioEncoder += "Motore".M[#K_MotoreInt].Out.SpazioCicloEnc;
	                            "Motore".M[#K_MotoreInt].Dati.ChFol_SpazioTarget += "Motore".M[#K_MotoreInt].Dati.TrgPosDint - "Motore".M[#K_MotoreInt].Dati.OldTrgPosDint;
	                            "Motore".M[#K_MotoreInt].Dati.ContCheckFollowError += REAL_TO_INT("Zona".Comuni.TempoCicloCpu_r);
	                        END_IF;
	                        "Motore".M[#K_MotoreInt].Dati.OldTrgPosDint := "Motore".M[#K_MotoreInt].Dati.TrgPosDint;
	                        IF "Motore".M[#K_MotoreInt].Prm.FollowingLimit > 0 AND NOT "Motore".M[#K_MotoreInt].Prm.Mech.EndLess THEN
	                            IF ABS("Motore".M[#K_MotoreInt].Out.FollowingError) > "Motore".M[#K_MotoreInt].Prm.FollowingLimit THEN
	                                "Motore".M[#K_MotoreInt].Allarmi.FolError := true;
	                            END_IF;
	                        END_IF;
	                    ELSE
	                        "Motore".M[#K_MotoreInt].Dati.ContCheckFollowError := 0;
	                        "Motore".M[#K_MotoreInt].Dati.ChFol_SpazioEncoder := "Motore".M[#K_MotoreInt].Dati.ChFol_SpazioTarget := 0;
	                    END_IF;
	                END_REGION
	                REGION Allarme direzione inversione
	                    IF NOT "Motore".M[#K_MotoreInt].Allarmi.Direzione THEN
	                        IF "Motore".M[#K_MotoreInt].Out.ActDirPos THEN
	                            "Motore".M[#K_MotoreInt].Dati.MemoCheckInversione += "Motore".M[#K_MotoreInt].Out.SpazioCicloEnc;
	                            IF "Motore".M[#K_MotoreInt].Dati.MemoCheckInversione > 0 THEN
	                                "Motore".M[#K_MotoreInt].Dati.MemoCheckInversione := 0;
	                            END_IF;
	                            IF "Motore".M[#K_MotoreInt].Dati.MemoCheckInversione < - #AppoMoltPrecisione THEN
	                                "Motore".M[#K_MotoreInt].Allarmi.Direzione := true;
	                            END_IF;
	                        ELSIF "Motore".M[#K_MotoreInt].Out.ActDirNeg THEN
	                            "Motore".M[#K_MotoreInt].Dati.MemoCheckInversione += "Motore".M[#K_MotoreInt].Out.SpazioCicloEnc;
	                            IF "Motore".M[#K_MotoreInt].Dati.MemoCheckInversione < 0 THEN
	                                "Motore".M[#K_MotoreInt].Dati.MemoCheckInversione := 0;
	                            END_IF;
	                            IF "Motore".M[#K_MotoreInt].Dati.MemoCheckInversione > #AppoMoltPrecisione THEN
	                                "Motore".M[#K_MotoreInt].Allarmi.Direzione := true;
	                            END_IF;
	                        ELSE
	                            "Motore".M[#K_MotoreInt].Dati.MemoCheckInversione := 0;
	                        END_IF;
	                    END_IF;
	                END_REGION
	                REGION Allarme Encoder Mismatch
	                    // L'allarme viene generato tutte le volte che l'encoder conta 10 volte la precisione nella dirazione non aspettata.
	                    IF "Motore".M[#K_MotoreInt].Dati.MotoreFermo AND "Motore".M[#K_MotoreInt].Dati.RitAggancioFreno THEN
	                        IF NOT "Motore".M[#K_MotoreInt].Dati.AppoImpMotoreFermo THEN
	                            "Motore".M[#K_MotoreInt].Dati.AppoImpMotoreFermo := true;
	                            "Motore".M[#K_MotoreInt].Dati.PosizioneAlloStop := "Motore".M[#K_MotoreInt].Out.ActPos;
	                        ELSIF ABS("Motore".M[#K_MotoreInt].Out.ActPos - "Motore".M[#K_MotoreInt].Dati.PosizioneAlloStop) > #AppoMoltPrecisione THEN
	                            "Motore".M[#K_MotoreInt].Allarmi.EncMismatch := true;
	                        END_IF;
	                    ELSE
	                        "Motore".M[#K_MotoreInt].Dati.AppoImpMotoreFermo := false;
	                    END_IF;
	                END_REGION
	                REGION Time Out Movimento Motore
	                    IF #FunzPositioning THEN
	                        IF NOT "Motore".M[#K_MotoreInt].Dati.AppoImpFunzPositioning THEN
	                            #ReqRicTempoProfilo := true;
	                        ELSIF #ReqCambioVel AND NOT "Motore".M[#K_MotoreInt].Dati.AppoImpCaVelPunto THEN
	                            #ReqRicTempoProfilo := true;
	                        ELSE
	                            #ReqRicTempoProfilo := #CambioReqAcc OR #CambioReqDec OR #CambioReqVel OR #REQSetup OR "Motore".M[#K_MotoreInt].Out.TrgPosFiltrata <> "Motore".M[#K_MotoreInt].Dati.TRG_OLD_POS_Select;
	                        END_IF;
	                        "Motore".M[#K_MotoreInt].Dati.AppoImpCaVelPunto := #ReqCambioVel;
	                        IF #ReqRicTempoProfilo THEN
	                            "Motore".M[#K_MotoreInt].Dati.TRG_OLD_POS_Select := "Motore".M[#K_MotoreInt].Out.TrgPosFiltrata;
	                            IF #ReqCambioVel THEN
	                                #VeloProfilo := "Motore".M[#K_MotoreInt].Dati.VeloDopoCambioRich;
	                            ELSE
	                                #VeloProfilo := "Motore".M[#K_MotoreInt].Dati.VeloRichPerc;
	                            END_IF;
	                            // Calcolo il tempo per la decelerazione
	                            IF #VeloProfilo > #VeloBassaConv THEN
	                                #TempoDec_Iniziale := (#VeloProfilo - #VeloBassaConv) / DINT_TO_REAL("Motore".M[#K_MotoreInt].Dati.DecReqInLavo);
	                            ELSE
	                                #TempoDec_Iniziale := 0.0;
	                            END_IF;
	                            // Tempo Decelerazione Finale
	                            #TempoDec_Finale := #VeloBassaConv / DINT_TO_REAL("Motore".M[#K_MotoreInt].Dati.DecReqFinaleInLavo);
	                            // Tempo accelerazione
	                            #TempoAcc := #VeloProfilo / DINT_TO_REAL("Motore".M[#K_MotoreInt].Dati.AccRichPerc);
	                            // Tempo a velocitÃ  fissa
	                            #TempoVFix := DINT_TO_REAL(#DistTRG_ASS) / #VeloProfilo;
	                            // Calcolo il tempo rimanente per l'esecuzione del profilo
	                            "Motore".M[#K_MotoreInt].Out.TFineProfilo := TRUNC((#TempoDec_Iniziale + #TempoDec_Finale + #TempoAcc + #TempoVFix) * 1000.0) + "Motore".M[#K_MotoreInt].Prm.TBassaVel + "Motore".M[#K_MotoreInt].Prm.TReazioneSistema;
	                            "Motore".M[#K_MotoreInt].Dati.ContTimeOutMovimento := 0;
	                            "Motore".M[#K_MotoreInt].Dati.TempoEsecuzioneProfilo := MAX(IN1 := "Motore".M[#K_MotoreInt].Out.TFineProfilo * 3, IN2 := 10000);
	                        END_IF;
	                        IF "Motore".M[#K_MotoreInt].Out.InMarcia THEN
	                            IF "Motore".M[#K_MotoreInt].Dati.ContTimeOutMovimento > "Motore".M[#K_MotoreInt].Dati.TempoEsecuzioneProfilo THEN
	                                "Motore".M[#K_MotoreInt].Allarmi.TOUTMovimento := true;
	                            ELSE
	                                "Motore".M[#K_MotoreInt].Dati.ContTimeOutMovimento += REAL_TO_INT("Zona".Comuni.TempoCicloCpu_r);
	                            END_IF;
	                        END_IF;
	                        "Motore".M[#K_MotoreInt].Dati.AppoImpFunzPositioning := true;
	                    ELSE
	                        "Motore".M[#K_MotoreInt].Dati.AppoImpFunzPositioning := false;
	                    END_IF;
	                END_REGION
	            END_IF;
	        END_REGION
	        REGION Gestione del Time Out Ricerca Sensore Azzeramento
	            // Nel caso di una richiesta di esecuzione di SetUP sul sensore
	            IF #SetUpSuSensore THEN
	                IF #REQSetupPannello AND NOT "Motore".M[#K_MotoreInt].Dati.SetupSensoreTrovato AND ("Motore".M[#K_MotoreInt].Out.ActDirPos OR "Motore".M[#K_MotoreInt].Out.ActDirNeg) THEN
	                    IF ("Motore".M[#K_MotoreInt].In.SensAzz AND "Motore".M[#K_MotoreInt].Dati.ContTimeOutAzzeramento > 5000) OR "Motore".M[#K_MotoreInt].Dati.ContTimeOutAzzeramento > 25000 THEN
	                        "Motore".M[#K_MotoreInt].Allarmi.TOUT_Azzeramento := TRUE;
	                    END_IF;
	                ELSE
	                    "Motore".M[#K_MotoreInt].Dati.ContTimeOutAzzeramento := 0;
	                END_IF;
	            ELSE
	                "Motore".M[#K_MotoreInt].Dati.ContTimeOutAzzeramento := 0;
	            END_IF;
	        END_REGION
	        REGION ALLARME: Time-Out Anticaduta
	            IF "Motore".M[#K_MotoreInt].Prm.AnticadutaPresente THEN
	                IF "Zona".Z[#K_Zona].Out.CentralinaOk THEN
	                    "Motore".M[#K_MotoreInt].Prm.ByPassAnticaduta := false;
	                END_IF;
	                "Motore".M[#K_MotoreInt].Out.CmdAnticaduta := ("Motore".M[#K_MotoreInt].Out.InMarcia AND "Motore".M[#K_MotoreInt].Out.CmdAnticaduta OR "Zona".Z[#K_Zona].Out.CentralinaOk) AND NOT "Motore".M[#K_MotoreInt].Out.DisContattori AND NOT "Motore".M[#K_MotoreInt].In.CinghiaRotta;
	                IF "Motore".M[#K_MotoreInt].Out.CmdAnticaduta AND NOT "Motore".M[#K_MotoreInt].In.AnticadutaON (*OR
	            NOT "Motor".M[#MotorNumber].o.CmdAnticaduta AND NOT "Motor".M[#MotorNumber].i.AnticadutaOFF*)THEN
	                    IF "Motore".M[#K_MotoreInt].Dati.ContTOutAnticaduta > 4000 THEN
	                        "Motore".M[#K_MotoreInt].Allarmi.TimeOutAnticaduta := true;
	                    ELSE
	                        "Motore".M[#K_MotoreInt].Dati.ContTOutAnticaduta += REAL_TO_INT("Zona".Comuni.TempoCicloCpu_r);
	                    END_IF;
	                ELSE
	                    "Motore".M[#K_MotoreInt].Dati.ContTOutAnticaduta := 0;
	                END_IF;
	            END_IF;
	        END_REGION
	        REGION Allarmi Generale Motore
	            "Motore".M[#K_MotoreInt].Allarmi.SezAperto := "Motore".M[#K_MotoreInt].In.SezAperto;
	            IF "Zona".Z[#K_Zona].Out.CentralinaOk THEN
	                IF "Motore".M[#K_MotoreInt].In.DriverFault THEN
	                    IF NOT "Motore".M[#K_MotoreInt].Dati.AlmInv_ResetInverter THEN
	                        IF "Motore".M[#K_MotoreInt].Dati.AlmInv_Cont >= "NResetInverter" THEN
	                            "Motore".M[#K_MotoreInt].Allarmi.InverterFault := true;
	                        ELSE
	                            "Motore".M[#K_MotoreInt].Dati.AlmInv_ContStorico += 1;
	                            "Motore".M[#K_MotoreInt].Dati.AlmInv_Cont += 1;
	                            "Motore".M[#K_MotoreInt].Dati.AlmInv_StoricoCodici["Motore".M[#K_MotoreInt].Dati.AlmInv_ContStorico MOD 10] := "Motore".M[#K_MotoreInt].HMI.CodiceAllarme;
	                            "Motore".M[#K_MotoreInt].Dati.MotorStop := true;
	                            "Motore".M[#K_MotoreInt].Dati.AlmInv_ResetInverter := true;
	                            "Motore".M[#K_MotoreInt].Dati.AlmInv_ToutReset := 0;
	                        END_IF;
	                    END_IF;
	                END_IF;
	                "Motore".M[#K_MotoreInt].Allarmi.InverterWarning := "Motore".M[#K_MotoreInt].In.DriverWarning;
	            END_IF;
	            IF "Motore".M[#K_MotoreInt].Dati.AlmInv_ResetInverter THEN
	                IF NOT "Motore".M[#K_MotoreInt].In.DriverFault THEN
	                    "Motore".M[#K_MotoreInt].Dati.AlmInv_ResetInverter := false;
	                END_IF;
	                "Motore".M[#K_MotoreInt].Dati.AlmInv_ToutReset += REAL_TO_INT("Zona".Comuni.TempoCicloCpu_r);
	                IF "Motore".M[#K_MotoreInt].Dati.AlmInv_ToutReset > 5000 THEN
	                    "Motore".M[#K_MotoreInt].Dati.AlmInv_ResetInverter := false;
	                    "Motore".M[#K_MotoreInt].Allarmi.InverterFault := true;
	                END_IF;
	            ELSE
	                "Motore".M[#K_MotoreInt].Dati.AlmInv_ToutReset := 0;
	            END_IF;
	            IF "Motore".M[#K_MotoreInt].In.NoComunInv THEN
	                "Motore".M[#K_MotoreInt].Allarmi.ComunInverter := true;
	            END_IF;
	            IF "Motore".M[#K_MotoreInt].In.NoComunEnc THEN
	                "Motore".M[#K_MotoreInt].Allarmi.ComunEncoder := true;
	            END_IF;
	            IF "Motore".M[#K_MotoreInt].In.TerVentolaOff THEN
	                "Motore".M[#K_MotoreInt].Allarmi.TermicoVentola := true;
	            END_IF;
	            IF "Motore".M[#K_MotoreInt].In.CinghiaRotta THEN
	                "Motore".M[#K_MotoreInt].Allarmi.RotturaCinghia := true;
	            END_IF;
	            IF "Motore".M[#K_MotoreInt].In.SpinaSicNoInPos THEN
	                "Motore".M[#K_MotoreInt].Allarmi.SpinaSicNoInPos := true;
	            END_IF;
	        END_REGION

	        REGION Conteggi Manutenzione Preventiva
	            IF "Motore".M[#K_MotoreInt].Prm.AbiltManutenzionePrev THEN
	                IF NOT "Motore".M[#K_MotoreInt].Dati.MotoreFermo THEN
	                    "Motore".M[#K_MotoreInt].Dati.MP.SpazioPercorso += ABS(IN := "Motore".M[#K_MotoreInt].Out.SpazioCicloEnc);
	                    IF "Motore".M[#K_MotoreInt].Dati.MP.SpazioPercorso > 1000000 THEN
	                        "Motore".M[#K_MotoreInt].Dati.MP.MetriPercorsi += 1;
	                        "Motore".M[#K_MotoreInt].Dati.MP.SpazioPercorso -= 1000000;
	                    END_IF;
	                    "Motore".M[#K_MotoreInt].Dati.MP.TempoMovimento += REAL_TO_INT("Zona".Comuni.TempoCicloCpu_r);
	                    IF "Motore".M[#K_MotoreInt].Dati.MP.TempoMovimento > 60000 THEN
	                        "Motore".M[#K_MotoreInt].Dati.MP.MinutiLavorati += 1;
	                        "Motore".M[#K_MotoreInt].Dati.MP.TempoMovimento -= 60000;
	                    END_IF;
	                    IF NOT "Motore".M[#K_MotoreInt].Dati.MP.ImpMarcia THEN
	                        "Motore".M[#K_MotoreInt].Dati.MP.NAvviamenti += 1;
	                        "Motore".M[#K_MotoreInt].Dati.MP.ImpMarcia := true;
	                    END_IF;
	                ELSE
	                    "Motore".M[#K_MotoreInt].Dati.MP.ImpMarcia := false;
	                END_IF;
	                IF "Motore".M[#K_MotoreInt].Out.CmdFreno AND NOT "Motore".M[#K_MotoreInt].Dati.MP.ImpFreno THEN
	                    "Motore".M[#K_MotoreInt].Dati.MP.NSgancioFreno += 1;
	                END_IF;
	                "Motore".M[#K_MotoreInt].Dati.MP.ImpFreno := "Motore".M[#K_MotoreInt].Out.CmdFreno;
	            END_IF;
	        END_REGION
	        REGION StatoMotoreHMI
	            (* Stati Motore
	            0 = Fermo
	            1 = Disabilitato da Area Automatico
	            2 = In allarme
	            3 = Disabilitato per motivi interni
	            4 = In premagnetizzazione con freno chiuso
	            5 = In premagnetizzazione con freno aperto
	            6 = In movimento positivo
	            7 = In movimento negativo
	            14 = In premagnetizzazione con freno chiuso con Allarme Attivo
	            15 = In premagnetizzazione con freno aperto con Allarme Attivo
	            16 = In movimento positivo con Allarme Attivo
	            17 = In movimento negativo con Allarme Attivo
	            20 = Dai Trasporti selezionato "Sempre fermo"
	            21 = Dai Trasporti selezionato "Sempre In Marcia Positivo"
	            22 = Dai Trasporti selezionato "Sempre In Marcia Negativo"
	            31 = Dai Trasporti selezionato "Sempre In Marcia Positivo" con Allarme Attivo
	            32 = Dai Trasporti selezionato "Sempre In Marcia Negativo" con Allarme Attivo
	            *)
	            IF "Motore".M[#K_MotoreInt].Out.ActDirPos THEN
	                IF "Motore".M[#K_MotoreInt].Out.Allarme THEN
	                    "Motore".M[#K_MotoreInt].HMI.Stato := 21;
	                ELSE
	                    "Motore".M[#K_MotoreInt].HMI.Stato := 6;
	                END_IF;
	                IF "Motore".M[#K_MotoreInt].Out.Allarme THEN
	                    "Motore".M[#K_MotoreInt].HMI.Stato += 10;
	                END_IF;
	            ELSIF "Motore".M[#K_MotoreInt].Out.ActDirNeg THEN
	                IF "Motore".M[#K_MotoreInt].Allarmi.A["KAllMot_22(Word1_x6)"].Stato THEN
	                    "Motore".M[#K_MotoreInt].HMI.Stato := 22;
	                ELSE
	                    "Motore".M[#K_MotoreInt].HMI.Stato := 7;
	                END_IF;
	                IF "Motore".M[#K_MotoreInt].Out.Allarme THEN
	                    "Motore".M[#K_MotoreInt].HMI.Stato += 10;
	                END_IF;
	            ELSIF NOT "Motore".M[#K_MotoreInt].Dati.MotoreFermo THEN
	                IF "Motore".M[#K_MotoreInt].Out.RitSgancioFreno THEN
	                    "Motore".M[#K_MotoreInt].HMI.Stato := 5;
	                ELSE
	                    "Motore".M[#K_MotoreInt].HMI.Stato := 4;
	                END_IF;
	                IF "Motore".M[#K_MotoreInt].Out.Allarme THEN
	                    "Motore".M[#K_MotoreInt].HMI.Stato += 10;
	                END_IF;
	            ELSIF "Motore".M[#K_MotoreInt].Out.Allarme THEN
	                "Motore".M[#K_MotoreInt].HMI.Stato := 2;
	            ELSIF NOT "Zona".Z[#K_Zona].Out.CentralinaOk THEN
	                "Motore".M[#K_MotoreInt].HMI.Stato := 1;
	            ELSIF NOT "Motore".M[#K_MotoreInt].Out.Pronto THEN
	                "Motore".M[#K_MotoreInt].HMI.Stato := 3;
	            ELSE
	                "Motore".M[#K_MotoreInt].HMI.Stato := 0;
	                IF "Motore".M[#K_MotoreInt].Allarmi.A["KAllMot_23(Word1_x7)"].Stato THEN
	                    "Motore".M[#K_MotoreInt].HMI.Stato := 20;
	                END_IF;
	            END_IF;
	        END_REGION
	        REGION StatoComandoHMI
	            (* Stati Motore
	            0 = Nessuna Richiesta
	            1 = Richiesto Jog Positivo
	            2 = Richiesto Jog Negativo
	            3 = Richiesta Posizionamento Assoluto, motore giÃ  in posizione
	            4 = Richiesta Posizionamento Assoluto, motore dovrÃ  muoversi in direzione positiva
	            5 = Richiesta Posizionamento Assoluto, motore dovrÃ  muoversi in direzione negativa
	            6 = Richiesta Posizionamento Relativo, motore giÃ  in posizione
	            7 = Richiesta Posizionamento Relativo, motore dovrÃ  muoversi in direzione positiva
	            8 = Richiesta Posizionamento Relativo, motore dovrÃ  muoversi in direzione negativa
	            9 = Richiesta Premagnetizzazione Positiva
	            10= Richiesta Premagnetizzazione Negativa
	            *)
	            IF "Motore".M[#K_MotoreInt].In.CmdPosRich THEN
	                "Motore".M[#K_MotoreInt].HMI.ComandoRichiesto := 1;
	            ELSIF "Motore".M[#K_MotoreInt].In.CmdNegRich THEN
	                "Motore".M[#K_MotoreInt].HMI.ComandoRichiesto := 2;
	            ELSIF "Motore".M[#K_MotoreInt].In.Positioning THEN
	                IF "Motore".M[#K_MotoreInt].Out.RichMovPos THEN
	                    "Motore".M[#K_MotoreInt].HMI.ComandoRichiesto := 4;
	                ELSIF "Motore".M[#K_MotoreInt].Out.RichMovNeg THEN
	                    "Motore".M[#K_MotoreInt].HMI.ComandoRichiesto := 5;
	                ELSE
	                    "Motore".M[#K_MotoreInt].HMI.ComandoRichiesto := 3;
	                END_IF;
	                IF "Motore".M[#K_MotoreInt].In.PosRelativo THEN
	                    "Motore".M[#K_MotoreInt].HMI.ComandoRichiesto += 3;
	                END_IF;
	            ELSIF "Motore".M[#K_MotoreInt].In.Premagnetizza THEN
	                IF "Motore".M[#K_MotoreInt].In.PremagnetizzaPos THEN
	                    "Motore".M[#K_MotoreInt].HMI.ComandoRichiesto := 9;
	                ELSIF "Motore".M[#K_MotoreInt].In.PremagnetizzaNeg THEN
	                    "Motore".M[#K_MotoreInt].HMI.ComandoRichiesto := 10;
	                ELSIF "Motore".M[#K_MotoreInt].Out.RichMovPos THEN
	                    "Motore".M[#K_MotoreInt].HMI.ComandoRichiesto := 9;
	                ELSIF "Motore".M[#K_MotoreInt].Out.RichMovNeg THEN
	                    "Motore".M[#K_MotoreInt].HMI.ComandoRichiesto := 10;
	                END_IF;
	            ELSE
	                "Motore".M[#K_MotoreInt].HMI.ComandoRichiesto := 0;
	            END_IF;
	        END_REGION
	    END_REGION ;
	    REGION To inverter
	        CASE "Motore".M[#K_MotoreInt].HW.TipoCollInverter OF
	            0:
	                REGION Inverter Comandato in Analogica
	                    "Motore".M[#K_MotoreInt].Out.Paw := DINT_TO_WORD(TRUNC("Motore".M[#K_MotoreInt].Out.VelAss / DINT_TO_REAL("Motore".M[#K_MotoreInt].Prm.C.VelMax) * DINT_TO_REAL("Motore".M[#K_MotoreInt].Prm.ValMaxRef)));
	                END_REGION ;
	            1:
	                REGION PN Mitsubishi
	                    (* Struttura Control Word
	                    Bit 00: Drive PO: Switch ON
	                    Bit 01: Drive PO: Output Shutoff Release
	                    Bit 02: Drive PO: Emergency Stop
	                    Bit 03: Drive PO: Enable
	                    Bit 04: Drive PO: Not Used
	                    Bit 05: Drive PO: Set Frequency Not retained
	                    Bit 06: Drive PO: Enble Set Point
	                    Bit 07: Drive PO: Fault Ack
	                    Bit 08: Drive PO: Not Used
	                    Bit 09: Drive PO: Used
	                    Bit 10: Drive PO: Comunication Enabled
	                    Bit 11: Drive PO: Target Torque Enabled
	                    Bit 12: Drive PO: Reverse Rotation
	                    Bit 13: Drive PO: Not Used
	                    Bit 14: Drive PO: Not Used
	                    Bit 15: Drive PO: Not Used
	                    *)
	                    #PO_Mitsubishi.CTW := w#16#200;
	                    #PO_Mitsubishi.CTW.%X0 := ("Motore".M[#K_MotoreInt].Out.CmdPosMotore OR "Motore".M[#K_MotoreInt].Out.CmdNegMotore) AND #PI_Mitsubishi.STW.%X0;
	                    #PO_Mitsubishi.CTW.%X1 := #PO_Mitsubishi.CTW.%X2 := "Zona".Z[#K_Zona].Out.CentralinaOk;
	                    #PO_Mitsubishi.CTW.%X3 := TRUE;
	                    #PO_Mitsubishi.CTW.%X5 := #PO_Mitsubishi.CTW.%X6 := true;
	                    #PO_Mitsubishi.CTW.%X12 := "Motore".M[#K_MotoreInt].Out.CmdNegMotore AND #PI_Mitsubishi.STW.%X0;
	                    #PO_Mitsubishi.CTW.%X7 := ("Zona".Z[#K_Zona].Gen.Reset OR ("Motore".M[#K_MotoreInt].Dati.AlmInv_ToutReset > 2000 AND "Zona".Comuni.Clocks.Clock1Hz)) AND "Motore".M[#K_MotoreInt].In.DriverFault;
	                    #PO_Mitsubishi.CTW.%X10 := true;
	                    #PO_Mitsubishi.Speed_SP := DINT_TO_INT(TRUNC("Motore".M[#K_MotoreInt].Out.VelAss / DINT_TO_REAL("Motore".M[#K_MotoreInt].Prm.C.VelMax) * 16384.0));
	                    #PO_Mitsubishi.Acc := TRUNC(DINT_TO_REAL("Motore".M[#K_MotoreInt].Prm.C.VelMax) / DINT_TO_REAL("Motore".M[#K_MotoreInt].Dati.AccRichPerc) * 3.0);
	                    #PO_Mitsubishi.Dec := TRUNC(DINT_TO_REAL("Motore".M[#K_MotoreInt].Prm.C.VelMax) / DINT_TO_REAL("Motore".M[#K_MotoreInt].Dati.DecReqInLavo) * 3.0);
	                    #PO_Mitsubishi.FStart := #VeloFrenoDir * 9000 / "Motore".M[#K_MotoreInt].Prm.C.VelMax;
	                    "Motore".M[#K_MotoreInt].Dati.RetVal_SCR_Inv := DPWR_DAT(LADDR := "Motore".M[#K_MotoreInt].HW.HWIO_Inverter, RECORD := #PO_Mitsubishi);
	                    "Motore".M[#K_MotoreInt].HMI.CTW1 := #PO_Mitsubishi.CTW;
	                END_REGION
	            2:
	                REGION PN Siemens
	                    (* Struttura Control Word
	                    Bit 00: Drive PO: Run = 1/Stop = 0
	                    Bit 01: Drive PO: Pulse Enable = 1/Pulse Disable = 0
	                    Bit 02: Drive PO: No Quick Stop = 1/Quick Stop = 0
	                    Bit 03: Drive PO: Enable = 1/Disable = 0
	                    Bit 04: Drive PO: Ramp Generator Enable = 1/Disable = 0
	                    Bit 05: Drive PO: Ramp Generator Unfreeze = 1/Freeze = 0
	                    Bit 06: Drive PO: Setpoint Enable = 1/ Disable = 0
	                    Bit 07: Drive PO: Faults/Warnings Acknowledge
	                    Bit 08: Drive PO: Reserved
	                    Bit 09: Drive PO: Reserved
	                    Bit 10: Drive PO: PLC Control
	                    Bit 11: Drive PO: Setpoint Reverse
	                    Bit 12: Drive PO: Reserved
	                    Bit 13: Drive PO: Motor Potentiometer Up
	                    Bit 14: Drive PO: Motor Potentiometer Down
	                    Bit 15: Drive PO: Reserved
	                    *)
	                    #PO_Siemens.CTW := w#16#47f;
	                    #PO_Siemens.CTW.%X0 := "Motore".M[#K_MotoreInt].Out.CmdPosMotore OR "Motore".M[#K_MotoreInt].Out.CmdNegMotore;
	                    #PO_Siemens.CTW.%X11 := "Motore".M[#K_MotoreInt].Out.CmdNegMotore;
	                    #PO_Siemens.CTW.%X7 := "Zona".Z[#K_Zona].Gen.Reset;
	                    #PO_Siemens.Speed := DINT_TO_INT(TRUNC("Motore".M[#K_MotoreInt].Out.VelAss / DINT_TO_REAL("Motore".M[#K_MotoreInt].Prm.C.VelMax) * 16384.0));
	                    "Motore".M[#K_MotoreInt].Dati.RetVal_SCR_Inv := DPWR_DAT(LADDR := "Motore".M[#K_MotoreInt].HW.HWIO_Inverter, RECORD := #PO_Siemens);
	                    "Motore".M[#K_MotoreInt].HMI.CTW1 := #PO_Siemens.CTW;
	                END_REGION
	            3:
	                REGION PN Schneider
	                    (* Struttura Control Word
	                    Bit 00: Switched on operating state; voltage at the power is enabled.
	                    Bit 01: 1= Coast Stop (OFF2) not active.
	                    Bit 02: 1 = Quick Stop (OFF3) not active.
	                    Bit 03: Enable electronics and pulses. The drive then runs-up to the reference frequency.
	                    Bit 04: Reserved
	                    Bit 05: Reserved
	                    Bit 06: Not used
	                    Bit 07: The fault reset function is active with a positive edge.
	                    Bit 08: Not used
	                    Bit 09: Not used
	                    Bit 10: Channel for the reference frequency and the command from the bus are active.
	                    Bit 11: Reserved
	                    Bit 12: Reserved
	                    Bit 13: Reserved
	                    Bit 14: Reserved
	                    Bit 15: Reserved
	                    *)
	                    #PO_Schneider.CTW := 0;
	                    #PO_Schneider.CTW.%X0 := #PI_Schneider.STW.%X0;
	                    // Normal Stop
	                    #PO_Schneider.CTW.%X1 := #PO_Schneider.CTW.%X2 := "Zona".Z[#K_Zona].Out.CentralinaOk AND NOT #PI_Schneider.STW.%X3;
	                    // Comando Marcia
	                    #PO_Schneider.CTW.%X3 := #PO_Schneider.CTW.%X0 AND ("Motore".M[#K_MotoreInt].Out.CmdPosMotore OR "Motore".M[#K_MotoreInt].Out.CmdNegMotore);
	                    //    Fault Reset
	                    #PO_Schneider.CTW.%X7 := "Zona".Z[#K_Zona].Gen.Reset AND #PI_Schneider.STW.%X3;
	                    // VelocitÃ  richiesta
	                    IF NOT "Motore".M[#K_MotoreInt].Out.CmdNegMotore THEN
	                        #PO_Schneider.Speed_SP := DINT_TO_INT(TRUNC("Motore".M[#K_MotoreInt].Out.VelAss / DINT_TO_REAL("Motore".M[#K_MotoreInt].Prm.C.VelMax) * 3000.0));
	                    ELSE
	                        #PO_Schneider.Speed_SP := - DINT_TO_INT(TRUNC("Motore".M[#K_MotoreInt].Out.VelAss / DINT_TO_REAL("Motore".M[#K_MotoreInt].Prm.C.VelMax) * 3000.0));
	                    END_IF;
	                    #PO_Schneider.Acc_SP := #PO_Schneider.Dec_SP := 0;
	                    "Motore".M[#K_MotoreInt].Dati.RetVal_SCR_Inv := DPWR_DAT(LADDR := "Motore".M[#K_MotoreInt].HW.HWIO_Inverter, RECORD := #PO_Schneider);
	                    "Motore".M[#K_MotoreInt].HMI.CTW1 := #PO_Schneider.CTW;
	                END_REGION
	            4:
	                REGION PN Movimot
	                    (* Struttura Control Word
	                    Bit 08: Reserved
	                    Bit 09: Reserved
	                    Bit 10: Reserved
	                    Bit 11: Reserved
	                    Bit 12: Reserved
	                    Bit 13: Reserved
	                    Bit 14: Reserved
	                    Bit 15: Reserved
	                    Bit 00: Enable 01 Run Motor
	                    Bit 01: Enable 02 Run Motor
	                    Bit 02: Enable 03 Run Motor
	                    Bit 03: Reserved
	                    Bit 04: Reserved
	                    Bit 05: Reserved
	                    Bit 06: Reset
	                    Bit 07: Reserved
	                    *)
	                    #PO_Movimot.CTW.%X1 := #PO_Movimot.CTW.%X2 := "Motore".M[#K_MotoreInt].Out.CmdPosMotore OR "Motore".M[#K_MotoreInt].Out.CmdNegMotore;
	                    #PO_Movimot.CTW.%X6 := ("Zona".Z[#K_Zona].Gen.Reset OR ("Motore".M[#K_MotoreInt].Dati.AlmInv_ToutReset > 2000 AND "Zona".Comuni.Clocks.Clock1Hz));
	                    IF NOT "Motore".M[#K_MotoreInt].Out.CmdNegMotore THEN
	                        #PO_Movimot.Speed := DINT_TO_INT(TRUNC("Motore".M[#K_MotoreInt].Out.VelAss / DINT_TO_REAL("Motore".M[#K_MotoreInt].Prm.C.VelMax) * 16384.0));
	                    ELSE
	                        #PO_Movimot.Speed := - DINT_TO_INT(TRUNC("Motore".M[#K_MotoreInt].Out.VelAss / DINT_TO_REAL("Motore".M[#K_MotoreInt].Prm.C.VelMax) * 16384.0));
	                    END_IF;
	                    #PO_Movimot.AccRich := DINT_TO_INT(TRUNC(DINT_TO_REAL("Motore".M[#K_MotoreInt].Prm.C.VelMax) / DINT_TO_REAL("Motore".M[#K_MotoreInt].Prm.DecEmergenza) * 400.0));
	                    "Motore".M[#K_MotoreInt].Dati.RetVal_SCR_Inv := DPWR_DAT(LADDR := "Motore".M[#K_MotoreInt].HW.HWIO_Inverter, RECORD := #PO_Movimot);
	                    "Motore".M[#K_MotoreInt].HMI.CTW1 := #PO_Movimot.CTW;
	                    "Motore".M[#K_MotoreInt].HMI.CTW2 := INT_TO_WORD(#PO_Movimot.Speed);
	                    "Motore".M[#K_MotoreInt].HMI.CTW3 := INT_TO_WORD(#PO_Movimot.AccRich);
	                END_REGION
	            5:
	                REGION PN MoviGear

	                    (* Struttura Control Word
	                    Bit 00: Enable/Emergency Stop
	                    Bit 01: Enable/Application Stop
	                    Bit 02: Riservato
	                    Bit 03: Rilascio Freno
	                    Bit 04: Jog Positivo
	                    Bit 05: Jog Negativo
	                    Bit 06: Nuovo Movimento Relativo
	                    Bit 07: Strat/Stop
	                    Bit 08: Fault Reset
	                    Bit 09: Riservato
	                    Bit 10: Attiva Motore 2
	                    Bit 11: Riservato
	                    Bit 12: Disabilita Limiti
	                    Bit 13: Attiva Output Stage
	                    Bit 14: Attiva Stand By
	                    Bit 15: HandShake
	                    *)
	                    #PO_MoviGear.CTW := 0;
	                    // Emergenza OK
	                    #PO_MoviGear.CTW.%X0 := "Zona".Z[#K_Zona].Out.CentralinaOk;
	                    // Comando di Marcia
	                    #PO_MoviGear.CTW.%X7 := #PO_MoviGear.CTW.%X1 := "Motore".M[#K_MotoreInt].Out.CmdPosMotore OR "Motore".M[#K_MotoreInt].Out.CmdNegMotore;
	                    // Fault Reset
	                    #PO_MoviGear.CTW.%X8 := "Zona".Z[#K_Zona].Gen.Reset;
	                    // VelocitÃ  richiesta
	                    IF NOT "Motore".M[#K_MotoreInt].Out.CmdNegMotore THEN
	                        #PO_MoviGear.Target_Speed := DINT_TO_INT(TRUNC("Motore".M[#K_MotoreInt].Out.VelAss / DINT_TO_REAL("Motore".M[#K_MotoreInt].Prm.C.VelMax) * 3000.0));
	                    ELSE
	                        #PO_MoviGear.Target_Speed := - DINT_TO_INT(TRUNC("Motore".M[#K_MotoreInt].Out.VelAss / DINT_TO_REAL("Motore".M[#K_MotoreInt].Prm.C.VelMax) * 3000.0));
	                    END_IF;
	                    #PO_MoviGear.Acceleration := #PO_MoviGear.Deceleration := 30000;
	                    #PO_MoviGear."DO".%X0 := "Motore".M[#K_MotoreInt].Out.CmdUsc01Inv;
	                    #PO_MoviGear."DO".%X1 := "Motore".M[#K_MotoreInt].Out.CmdUsc02Inv;
	                    "Motore".M[#K_MotoreInt].Dati.RetVal_SCR_Inv := DPWR_DAT(LADDR := "Motore".M[#K_MotoreInt].HW.HWIO_Inverter, RECORD := #PO_MoviGear);
	                    "Motore".M[#K_MotoreInt].HMI.CTW1 := #PO_MoviGear.CTW;
	                END_REGION
	            6:
	                REGION PN Danfoss
	                    (* Struttura Control Word
	                       Bit 08: JOG 1 OFF/ON
	                       Bit 09: JOG 2 OFF/ON
	                       Bit 10: 0=Data invalid    1=Data valid
	                       Bit 11: 0=No function        1=Slow down
	                       Bit 12: 0=No function        1=Catch up
	                       Bit 13: 0=Parameter set-up        1=Sel LSB
	                       Bit 14: 0=Parameter set-up        1=Sel MSB
	                       Bit 15: 0=No function        1=Reserve
	                       Bit 00: OFF/ON 1
	                       Bit 01: OFF/ON 2
	                       Bit 02: OFF/ON 3
	                       Bit 03: 0=Coasting        1=Not coasting
	                       Bit 04: 0=Quick stop       1=Ramp
	                       Bit 05: 0=Hold Freq.Output   1=Use Ramp
	                       Bit 06: 0=Ramp Stop        1=Start
	                       Bit 07: 0=No function        1=Reset
	                       *)
	                    #PO_Danfoss.CTW := w#16#47f;
	                    #PO_Danfoss.CTW.%X0 := #PI_Danfoss.STW.%X0;
	                    #PO_Danfoss.CTW.%X6 := ("Motore".M[#K_MotoreInt].Out.CmdPosMotore OR "Motore".M[#K_MotoreInt].Out.CmdNegMotore) AND #PO_Danfoss.CTW.%X0 AND #PI_Danfoss.STW.%X9;
	                    #PO_Danfoss.CTW.%X15 := #PO_Danfoss.CTW.%X6 AND "Motore".M[#K_MotoreInt].Out.CmdNegMotore;
	                    #PO_Danfoss.CTW.%X7 := "Zona".Z[#K_Zona].Gen.Reset AND #PI_Danfoss.STW.%X3;
	                    #PO_Danfoss.Speed := DINT_TO_INT(TRUNC("Motore".M[#K_MotoreInt].Out.VelAss / DINT_TO_REAL("Motore".M[#K_MotoreInt].Prm.C.VelMax) * 16384.0));
	                    #PO_Danfoss.AccRich := DINT_TO_INT(TRUNC(DINT_TO_REAL("Motore".M[#K_MotoreInt].Prm.C.VelMax) / DINT_TO_REAL("Motore".M[#K_MotoreInt].Dati.AccRichPerc) * 40.0));
	                    #PO_Danfoss.DecRich := DINT_TO_INT(TRUNC(DINT_TO_REAL("Motore".M[#K_MotoreInt].Prm.C.VelMax) / DINT_TO_REAL(#DecActRich) * 40.0));
	                    "Motore".M[#K_MotoreInt].Dati.RetVal_SCR_Inv := DPWR_DAT(LADDR := "Motore".M[#K_MotoreInt].HW.HWIO_Inverter, RECORD := #PO_Danfoss);
	                    "Motore".M[#K_MotoreInt].HMI.CTW1 := #PO_Danfoss.CTW;
	                END_REGION ;
	            7:
	                REGION PN MoviTrak
	                    (* Struttura Control Word
	                    Bit 08: Reserved
	                    Bit 09: Reserved
	                    Bit 10: Reserved
	                    Bit 11: Reserved
	                    Bit 12: Reserved
	                    Bit 13: Reserved
	                    Bit 14: Reserved
	                    Bit 15: Reserved
	                    Bit 00: Inhibit/Enable
	                    Bit 01: Enable/Rapid Stop
	                    Bit 02: Enable/Stop
	                    Bit 03: Reserved
	                    Bit 04: Reserved
	                    Bit 05: Reserved
	                    Bit 06: Reset
	                    Bit 07: Reserved
	                    *)
	                    #PO_MoviTrac.CTW := 0;
	                    #PO_MoviTrac.CTW.%X1 := #PO_MoviTrac.CTW.%X2 := "Motore".M[#K_MotoreInt].Out.CmdPosMotore OR "Motore".M[#K_MotoreInt].Out.CmdNegMotore;
	                    #PO_MoviTrac.CTW.%X6 := "Zona".Z[#K_Zona].Gen.Reset;
	                    IF NOT "Motore".M[#K_MotoreInt].Out.CmdNegMotore THEN
	                        #PO_MoviTrac.Speed := DINT_TO_INT(TRUNC("Motore".M[#K_MotoreInt].Out.VelAss / DINT_TO_REAL("Motore".M[#K_MotoreInt].Prm.C.VelMax) * 16384.0));
	                    ELSE
	                        #PO_MoviTrac.Speed := - DINT_TO_INT(TRUNC("Motore".M[#K_MotoreInt].Out.VelAss / DINT_TO_REAL("Motore".M[#K_MotoreInt].Prm.C.VelMax) * 16384.0));
	                    END_IF;
	                    "Motore".M[#K_MotoreInt].Dati.RetVal_SCR_Inv := DPWR_DAT(LADDR := "Motore".M[#K_MotoreInt].HW.HWIO_Inverter, RECORD := #PO_MoviTrac);
	                    "Motore".M[#K_MotoreInt].HMI.CTW1 := #PO_MoviTrac.CTW;
	                END_REGION
	            8:
	                REGION PN INVT
	                    (* Struttura Control Word
	                    Byte 0
	                    DEC Description
	                    1   Forward running
	                    2   Reverse running
	                    3   Forward inching
	                    4   Reverse inching
	                    5   Decelerating to stop
	                    6   Coasting to stop (emergency stop)
	                    7   Fault reset
	                    8   Jogging to stop
	                    9   Decelerate to stop
	                    ////////////////////////////////////////////////
	                    Bit 8: Abilita scrittura parametri PKW
	                    ////////////////////////////////////////////////
	                    Bit 9-10:
	                    DEC DEscrizione
	                    00  Motor 1
	                    01  Motor 2
	                    ////////////////////////////////////////////////
	                    Bit 11: 0=Disable Switchig, 1=Enable Torque/Speed control Switching
	                    Bit 12: Reset Power Consumption
	                    Bit 13: Pre-Excitation
	                    Bit 14: DC-Bracking
	                    Bit 15: Heart Beat Reference

